// SIMATIC S7-200 project (STEP 7-Micro/WIN), CPU 221 REL 01.10

SYMBOL_TABLE 用户定义1
启动               I0.0
东西灯G             Q0.0
东西灯Y             Q0.1
东西灯R             Q0.2
南北灯G             Q0.3
南北灯Y             Q0.4
南北灯R             Q0.5
定时器              T37
END_SYMBOL_TABLE

ORGANIZATION_BLOCK 主程序:OB1
TITLE=程序注释   十字路口交通灯控制
BEGIN
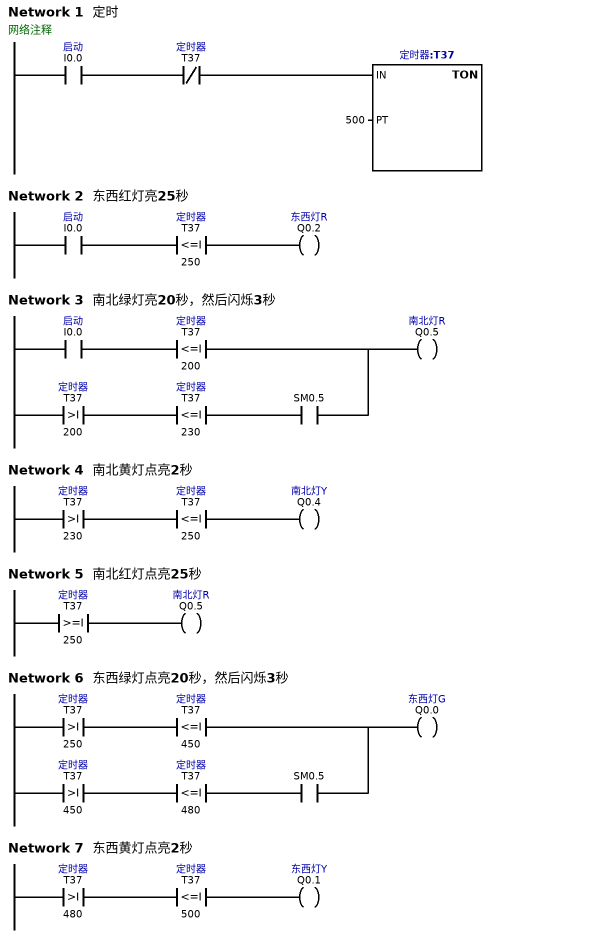
Network 1 // 定时
// 网络注释
LD     启动:I0.0
AN     定时器:T37
TON    定时器:T37, 500
Network 2 // 东西红灯亮25秒
LD     启动:I0.0
AW<=   定时器:T37, 250
=      东西灯R:Q0.2
Network 3 // 南北绿灯亮20秒，然后闪烁3秒
LD     启动:I0.0
AW<=   定时器:T37, 200
LDW>   定时器:T37, 200
AW<=   定时器:T37, 230
A      SM0.5
OLD
=      南北灯R:Q0.5
Network 4 // 南北黄灯点亮2秒
LDW>   定时器:T37, 230
AW<=   定时器:T37, 250
=      南北灯Y:Q0.4
Network 5 // 南北红灯点亮25秒
LDW>=  定时器:T37, 250
=      南北灯R:Q0.5
Network 6 // 东西绿灯点亮20秒，然后闪烁3秒
LDW>   定时器:T37, 250
AW<=   定时器:T37, 450
LDW>   定时器:T37, 450
AW<=   定时器:T37, 480
A      SM0.5
OLD
=      东西灯G:Q0.0
Network 7 // 东西黄灯点亮2秒
LDW>   定时器:T37, 480
AW<=   定时器:T37, 500
=      东西灯Y:Q0.1
END_ORGANIZATION_BLOCK
